{attribute 'qualified_only'}
{attribute 'strict'}
{attribute 'to_string'}
TYPE E_Trajectory :
(
    Sine := 0,
    Ramp := 1
);
END_TYPE

(* stored: Version 1.1.0.1
   DUT E_Trajectory: Id {1d98368d-1282-4545-95ff-91b5c985e7ba} *)
